{attribute 'enable_dynamic_creation'}
FUNCTION_BLOCK FutureMCInching EXTENDS FB_AbstructFuture
VAR_INPUT
END_VAR
VAR_OUTPUT
END_VAR
VAR
	_mc_jog	: MC_Jog;
	_mc_reset	: MC_Reset;
	_abort_executor		: FB_Executor;
	_axis: REFERENCE TO AXIS_REF;
	_direction : BOOL;
	_position : MC_LREAL;
	_velocity : MC_LREAL;
	_acceleration: MC_LREAL;
	_deceleration: MC_LREAL;
	_jerk		: MC_LREAL;
	_mode : E_JogMode ;
	_error_id :UDINT;
	_reset_state : UINT;
	step : UINT;
END_VAR

METHOD error_reset : BOOL // Must be overrided if future has any errors.
VAR_INST
	watch_delay  : TON;
END_VAR
_error_id := _mc_jog.ErrorID;
IF _error_id <> 0 THEN
	CASE _reset_state OF
		0:
			_mc_reset(Axis := _axis, Execute := FALSE);
			_mc_reset(Axis:= _axis, Execute := TRUE );
			watch_delay(IN := FALSE);
			_reset_state := 1;
		1:
			IF _mc_reset.Busy THEN
				_mc_reset(Axis:= _axis,Execute := FALSE);
				_reset_state := 2;
			END_IF
		2:
			IF _error_id = 0 THEN
				error_reset := TRUE;
				_reset_state := 0;
			ELSE
				watch_delay(IN := TRUE, PT := T#1S);
				IF watch_delay.Q THEN
					error_reset := TRUE;
					_reset_state := 0;
				END_IF
			END_IF
	END_CASE
	
	IF _error_id = 0 THEN
		_reset_state := 0;
	END_IF
ELSE
	error_reset := TRUE;
END_IF
END_METHOD

METHOD execute : BOOL // Return TRUE if finish.
CASE step OF
	0:
		_mc_jog(
			JogForward := _direction,
			JogBackwards := NOT _direction,
			Axis := _axis,
			Position := _position,
			Velocity := _velocity,
			Acceleration := _acceleration,
			Deceleration := _deceleration,
			Jerk := _jerk,
			Mode := E_JogMode.MC_JOGMODE_INCHING
		);
		IF _mc_jog.Done OR _mc_jog.Error THEN
			step := 1;
		END_IF

	1:
		_mc_jog(JogForward := FALSE, JogBackwards := FALSE, Axis := _axis);
		execute := TRUE;
		_error_id := _mc_jog.ErrorID;		
END_CASE
END_METHOD

METHOD init : BOOL // Return TRUE if finish.

VAR
	axis: INT;
END_VAR
_reset_state := 0;
_error_id := _mc_jog.ErrorID;
step := 0;
init := TRUE;
END_METHOD

PROPERTY nErrorID : UDINT
GET
nErrorID := _error_id;
END_GET
SET
END_SET
END_PROPERTY

METHOD set_options : BOOL
VAR_INPUT
	acceleration	: MC_LREAL;		// Set deceleration in case let moving axis halt.
	deceleration	: MC_LREAL;		// Set deceleration in case let moving axis halt.
	jerk			: MC_LREAL;		// Set jerk in case let moving axis halt.
END_VAR
_acceleration := acceleration;
_deceleration := deceleration;
_jerk := jerk;
END_METHOD

METHOD set_parameters : BOOL
VAR_INPUT
	axis : REFERENCE TO AXIS_REF;
	direction : BOOL;
	position : MC_LREAL;
	velocity : MC_LREAL;
END_VAR
_axis REF= axis;
_direction := direction;
_position := position;
_velocity := velocity;
END_METHOD

END_FUNCTION_BLOCK

(* stored: Version 1.1.0.1, ProductVersion 3.1.4024.15
   POU FutureMCInching: Id {2d0d01ce-3012-43a6-9be6-fc6a356527f7}, SpecialFunc None
   Method error_reset: Id {ba0c1137-f841-47ad-a273-1d21c49fdbdd}
   Method execute: Id {5af710ba-7d2f-4925-b8ea-ddc87569205a}
   Method init: Id {631c5c17-d70c-4519-a09b-d32b82adcea0}
   Property nErrorID: Id {b433b11e-449b-410e-af2f-363681da691e}
   Get Get: Id {c626f03a-dd6a-4e73-9760-b26289a6edf3}
   Set Set: Id {1e02bef9-7ff3-4433-ac1a-74e3b19fc7f9}
   Method set_options: Id {4df2ee6c-677d-4f34-a6c1-e171e6cf333e}
   Method set_parameters: Id {e9984d08-137c-4257-88d6-0495598af661} *)
